// TIA Portal V21 export
DATA_BLOCK "DB609"   // DB609
AUTHOR : PRECISE
FAMILY : PRECISE
// stored: AutoNumber false, InstanceOfName FB609, InstanceOfType FB
"FB609"
   // VAR_INPUT
   //    CipSelected : Bool;
   //    CycleEnable : Bool;
   //    CycleRunning : Bool;
   //    SecPulse : Bool;
   //    AlwaysTrue : Bool;
   //    ParaIn : "DrainInputs";
   //    ActualWeight : Real;
   //    ActualPressure : Real;
   //    ActualConductivityVessel : Real;
   //    ActualRepetition : Int;
   //    ActualSkidWeight : Real;
   // END_VAR
   // VAR_OUTPUT
   //    Started : Bool;
   //    PressureUtilityValve : Bool;
   //    "Line Valves" : Bool;
   //    ParaOut : "DrainOutputs";
   //    StepStatus : String[60];
   //    Print : "DrainPrint";
   //    PrintConductivityNotSampled : "ConductivityNotSampled";
   // END_VAR
   // VAR_IN_OUT
   //    Over : Bool;
   //    OverTemp : Bool;
   //    PressurePostiveTol : Real;
   //    PressureNegativeTol : Real;
   //    Temp1 : Int;
   //    Temp2 : Int;
   //    SampledConductivityVessel : Real;
   //    ConductivitySuccess : Bool;
   //    ConductivityNotSampled : Bool;
   //    RE1 : Bool;
   //    RE2 : Bool;
   //    RE3 : Bool;
   //    RE4 : Bool;
   //    RE5 : Bool;
   //    ControlStarted : Bool;
   //    SetPressureReached : Bool;
   //    DrainOverValve : Bool;
   //    ConductivityCheckBit : Bool;
   //    ActualConductivityPTL : Real;
   //    SampledConductivityPTL : Real;
   //    ConductivitySuccessVessel : Bool;
   //    ConductivitySuccessPtl : Bool;
   //    Temp3 : Int;
   //    Temp4 : Int;
   //    Temp5 : Int;
   //    Temp6 : Int;
   //    Temp7 : Int;
   //    Temp8 : Int;
   //    EndConfirmationPopupSel : Bool;
   //    EndConfirmationPopup : Bool;
   //    EndConfirmationPopupAck : Bool;
   //    RE_1 : Bool;
   //    TempBit : Bool;
   //    RE6 : Bool;
   // END_VAR
   // VAR
   //    ValveOnDelayPV : Int;
   //    ValveOffDelayPV : Int;
   //    StepDelay { S7_SetPoint := 'True'} : "FB110";
   //    ResetPrintValues { S7_SetPoint := 'True'} : TON_TIME;
   // END_VAR
BEGIN
END_DATA_BLOCK
